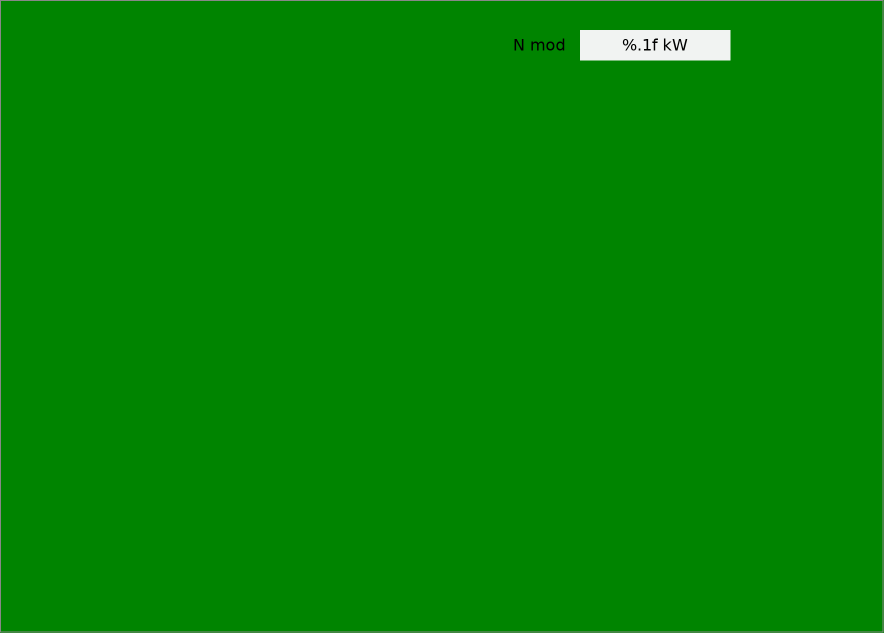
VISUALIZATION PM_config  // 884x633
    Rectangle (510,30 70x30), "N mod"
    Rectangle (580,30 150x30), "%.1f kW", text variable: GVL_CONV_COMMS.P_Measured[1]
END_VISUALIZATION

(* stored: Version 1.1.0.1, ProductVersion 3.1.4024.11
   Visu PM_config: Id {85103abf-7e7c-4998-be20-7e23a3fc5357} *)
